FUNCTION_BLOCK MoveGarageDoor
VAR_INPUT
	bActuationProgram : BOOL; //actuation button for moving the door
	bError : BOOL; //input error
END_VAR
VAR_OUTPUT
	bClosed : BOOL; //sensor that indicates whether or not the door is closed
	bOpened : BOOL; //sensor that indicates whether or not the door is opened
	bDriveOverload : BOOL; //sensor that indicates whether or not there is an error
	bPaused : BOOL; //sensor that indicates that the door is paused
	bLight : BOOL; //light that shows there is motion
	fActPos : LREAL; //actual position of the axis
	
	bVis1O : BOOL;
	bVis2O : BOOL;
	bVis3O : BOOL;
	bVis1C : BOOL;
	bVis2C : BOOL;
	bErrorImg : BOOL;
	bPauseImg : BOOL;

END_VAR
VAR
	bInitialActivate : BOOL; //helps set the door to closed at the start
	
	fbActivate : R_TRIG;
	fbInitial : R_TRIG; //helps set the initial value to closed
	
	bActuation : BOOL; //works with the actuation program inside of the function block
	
	iState : UDINT;
	
	Actuator : AXIS_REF; //we refrence the axis
	McPower : MC_Power; //power and reset function blocks for the axis
	McReset : MC_Reset;
	McMove : MC_MoveAbsolute;
	McStop : MC_Stop;

	
	bTempC : BOOL; //helps determine what was the door doing before pause/error
	bTempO : BOOL;
	
	fbBlinker : Blinker;
	

END_VAR

bInitialActivate := TRUE; //we close the door at the start
fbInitial(CLK := TRUE);
IF fbInitial.Q THEN
	bClosed := TRUE; //we have set the door to closed at the start (only activates the first time we run the program
END_IF

CASE iState OF
	0:	
		IF McPower.Status THEN
			iState := 10;
		END_IF
	5: //turning actuation off
		bActuation := FALSE;
		iState := 0; //return to the first state
	10:
		fbActivate(CLK := bActuationProgram);
		IF fbActivate.Q THEN
			bActuation := TRUE;
		END_IF
		bTempO := FALSE;
		bTempC := FALSE;
		IF bActuation THEN
			iState := 20; //if we click the button go to the next state and check it's state
		END_IF
	15:
		bActuation := FALSE;
		iState := 100;	
	20:
		IF bClosed THEN
			iState := 40; //open state
		ELSIF bOpened THEN
			iState := 50; //close state
		ELSE
			iState := 999;// driveoverload state
		END_IF
	30:
		bActuation := FALSE;
		iState := 999;
	40: //the door is closed we open it
		bClosed := FALSE;	
		IF bActuation THEN
			bLight := TRUE;
			bTempO := TRUE;
			McMove(Axis := Actuator, //we open the door (100 means openned)
					Position := 1000,
					Velocity := 100,
					Acceleration := 100,
					Deceleration := 100,
					Jerk := 100000,
					Execute := TRUE);
			iState := 45;	
		END_IF
	45:	//check if the movement is done
		fbActivate(CLK := bActuationProgram); //incase we want to pause it
		IF fbActivate.Q THEN
			bActuation := FALSE;
		END_IF
		IF bError THEN
			iState := 30; //incase the door goes to error
		END_IF
		IF bActuation THEN	
			IF McMove.Done AND NOT McMove.Error THEN
				McMove(Axis := Actuator,Execute := FALSE); //we turn it off
				bOpened := TRUE;
				bLight := FALSE;
				iState := 5;
			END_IF
		ELSE
			bPaused := TRUE;
			iState := 15;	
		END_IF
	50: //door is opened we close it
		bOpened := FALSE;	
		IF bActuation THEN
			bLight := TRUE;
			bTempC := TRUE;
			McMove(Axis := Actuator, //we close the door  (0 means openned)
					Position := 0,
					Velocity := 100,
					Acceleration := 100,
					Deceleration := 100,
					Jerk := 100000,
					Execute := TRUE);
			iState := 55; //check if the movement is done
		END_IF	
	55: //check if the movement is done
		fbActivate(CLK := bActuationProgram); //incase we want to pause it
		IF fbActivate.Q THEN
			bActuation := FALSE;
		END_IF
		IF bError THEN
			iState := 30; //incase the door goes to error
		END_IF
		IF bActuation THEN
			
	
			IF McMove.Done AND NOT McMove.Error THEN
				McMove(Axis := Actuator,Execute := FALSE); //we turn it off
				bClosed := TRUE;
				bLight := FALSE;
				iState := 5;
			END_IF
		ELSE
			bPaused := TRUE;
			iState := 15;	
		END_IF
		
	100: //pause state
		//bVis1O := FALSE;
		//bVis2O := FALSE;
		//bVis3O := FALSE;
		//bVis1C := FALSE;
		//bVis2C := FALSE;
		//bPauseImg := TRUE;
		
		bLight := FALSE;
		fbActivate(CLK := bActuationProgram);		
		IF fbActivate.Q THEN
			bActuation := TRUE;
			bPaused := FALSE; //we turn off the pause light
		END_IF
		McStop(Axis := Actuator,
				Deceleration := 300,
				Execute := TRUE);
		IF bActuation AND bTempC THEN
			bLight := TRUE;
			bTempC := FALSE;
			McStop(Axis := Actuator,Execute := FALSE);
			McMove(Axis := Actuator,Execute := FALSE);
			iState := 40;
		ELSIF bActuation AND bTempO THEN
			bLight := TRUE;
			bTempO := FALSE;
			McStop(Axis := Actuator,Execute := FALSE);
			McMove(Axis := Actuator,Execute := FALSE);
			iState := 50;	
		END_IF
				


	999: //error state	
		bErrorImg := TRUE;
		
		bLight := fbBlinker.bBlink;
		fbBlinker();
		bDriveOverload := TRUE;
		fbActivate(CLK := bActuationProgram);		
		IF fbActivate.Q THEN
			bActuation := TRUE;
			bPaused := FALSE; //we turn off the pause light
		END_IF
		McStop(Axis := Actuator,
				Deceleration := 300,
				Execute := TRUE);
		IF bActuation AND bTempC THEN
			bErrorImg := FALSE;
			bDriveOverload := FALSE;
			bLight := TRUE;
			bTempC := FALSE;
			McStop(Axis := Actuator,Execute := FALSE);
			McMove(Axis := Actuator,Execute := FALSE);
			iState := 40;
		ELSIF bActuation AND bTempO THEN
			bErrorImg := FALSE;
			bDriveOverload := FALSE;
			bLight := TRUE;
			bTempO := FALSE;
			McStop(Axis := Actuator,Execute := FALSE);
			McMove(Axis := Actuator,Execute := FALSE);
			iState := 50;	
		END_IF
		
END_CASE
Actuator.ReadStatus(); //referencing the axis to the function blocks
McPower(Axis := Actuator,Enable := TRUE,Enable_Positive := TRUE,Enable_Negative := TRUE);
McReset(Axis := Actuator);
McMove(Axis := Actuator);
McStop(Axis := Actuator);

fActPos := Actuator.NcToPlc.ActPos;

IF bTempO THEN
	//bErrorImg := FALSE;
	//bPauseImg := FALSE;
	bVis1C := FALSE;
	bVis2C := FALSE;
	IF fActPos > 180.0 THEN
		bVis1O := TRUE;
	END_IF
	IF fActPos > 550.0 THEN
		bVis2O := TRUE;
		bVis1O := FALSE;
	END_IF
	IF fActPos > 850.0 THEN
		bVis2O := FALSE;
		bVis3O := TRUE;
	END_IF
END_IF

IF bTempC THEN
	//bErrorImg := FALSE;
	//bPauseImg := FALSE;
	bVis1O := FALSE;
	bVis2O := FALSE;
	IF fActPos < 850.0 THEN
		bVis1C := TRUE;
		bVis3O := FALSE;
	END_IF
	IF fActPos < 550.0 THEN
		bVis2C := TRUE;
		bVis1C := FALSE;
	END_IF
	IF fActPos < 180.0 THEN
		bVis2C := FALSE;
	END_IF
END_IF

END_FUNCTION_BLOCK

(* stored: Version 1.1.0.1, ProductVersion 3.1.4024.12
   POU MoveGarageDoor: Id {bdd996a8-9082-46e2-b8c7-666d28e05c38}, SpecialFunc None *)
